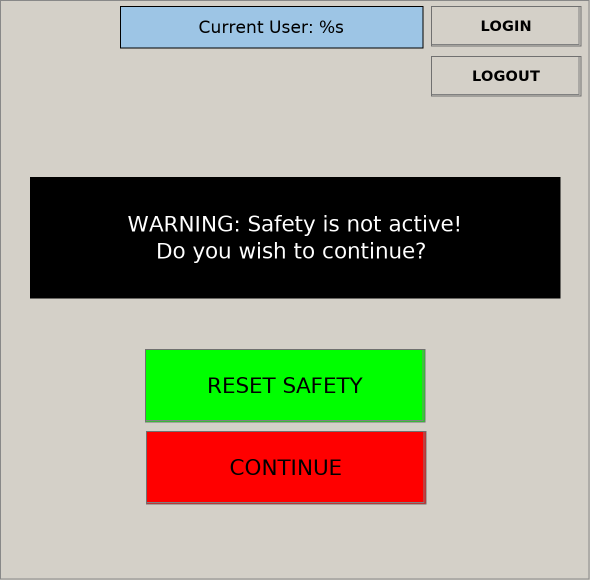
VISUALIZATION safetyDisableWarning  // 590x580
    Rectangle (30,177 530x121), "WARNING: Safety is not active! Do you wish to continue?", text variable: MAIN.sSafetyResetMsg
    Button (145,349 280x73), "RESET SAFETY"
        toggle GVL_machine.bSafetyBypass
    Button (146,431 280x73), "CONTINUE"
        OnMouseDown: change screen: Previous 
        OnMouseDown: execute { main.fbSafetyBypassTim(IN := FALSE); }
    Button (431,6 150x40), "LOGIN"
        OnMouseDown: VisuUserMgmt Type=Login
    Button (431,56 150x40), "LOGOUT"
        OnMouseDown: VisuUserMgmt Type=Logout
    Textfield (120,6 303x42), "Current User: %s", text variable: VisuElems.CurrentUserName
END_VISUALIZATION

// ---- VISUs/VISUs/safetyResetScreen.TcVIS
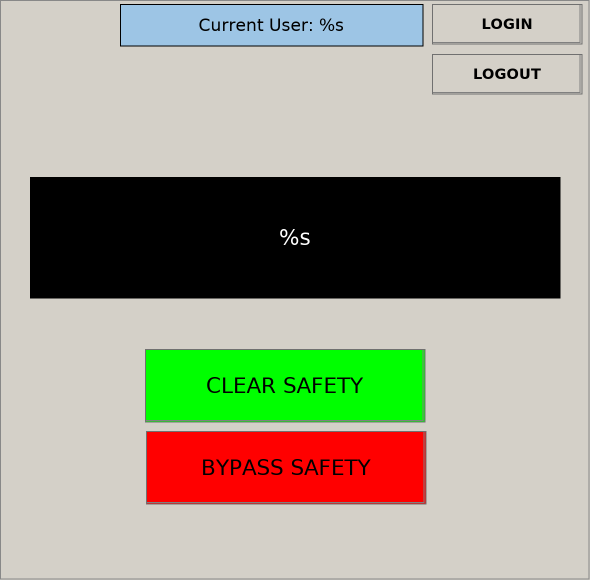
VISUALIZATION safetyResetScreen  // 590x580
    Rectangle (30,177 530x121), "%s", text variable: MAIN.sSafetyResetMsg
    Button (145,349 280x73), "CLEAR SAFETY"
        toggle MAIN.bSafetyResetBtn
    Button (146,431 280x73), "BYPASS SAFETY"
        toggle GVL_machine.bSafetyBypass
        OnMouseDown: execute {
            IF NOT GVL_devices.fbEstop.bEstopSigOk THEN
            	main.bBypassResetEstop := TRUE;
            END_IF
        }
    Button (432,4 150x40), "LOGIN"
        OnMouseDown: VisuUserMgmt Type=Login
    Button (432,54 150x40), "LOGOUT"
        OnMouseDown: VisuUserMgmt Type=Logout
    Textfield (120,4 303x42), "Current User: %s", text variable: VisuElems.CurrentUserName
END_VISUALIZATION

// ---- VISUs/VISUs/settingsScreen.TcVIS
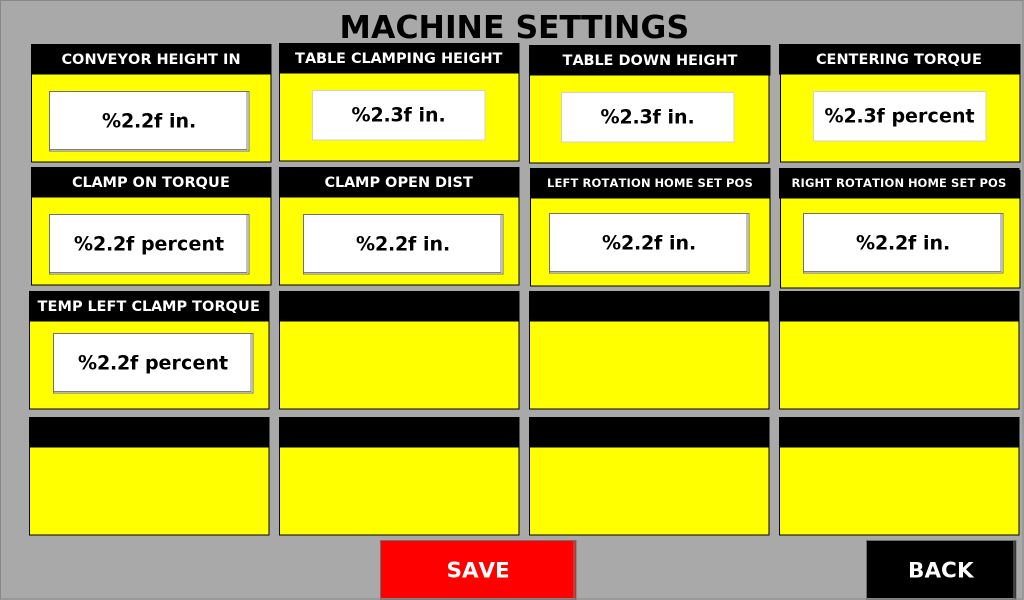
VISUALIZATION settingsScreen  // 1024x600
    RoundedRectangle (29,291 240x118)
    RoundedRectangle (279,43 240x118)
    RoundedRectangle (529,45 240x118)
    RoundedRectangle (29,417 240x118)
    RoundedRectangle (780,44 240x118)
    RoundedRectangle (780,170 240x118)
    RoundedRectangle (530,168 240x118)
    RoundedRectangle (279,291 240x118)
    RoundedRectangle (279,417 240x118)
    Label (183,10 663x34), "MACHINE SETTINGS"
    Textfield (661,76 61x30)
    Textfield (583,76 61x30)
    Textfield (327,202 61x30)
    Textfield (555,75 84x30)
    RoundedRectangle (279,417 240x30)
    RoundedRectangle (279,291 240x30)
    RoundedRectangle (29,291 240x30), "TEMP LEFT CLAMP TORQUE"
    RoundedRectangle (29,417 240x30)
    Textfield (680,76 61x30)
    Textfield (813,91 173x50), "%2.3f percent", text variable: GVL_persistent.fCenteringTorque
        OnMouseClick: write the text variable via VisuDialogs.Numpad
        OnMouseClick: OpenDialog Dialog=VisuDialogs.MessageBox, Parameters={eType: VisuDialogs.MessageBoxDialog_Types.OK, sMessageTxt: GVL_machine.sEditMessage, sTitle: GVL_machine.sEditTitle}, OpenModal=True, OpenCentered=True
        OnMouseClick: execute { GVL_machine.bFlashSaveBtn := TRUE; }
    Textfield (312,90 173x50), "%2.3f in.", text variable: GVL_persistent.fTableClampHeight
        OnMouseClick: write the text variable via VisuDialogs.Numpad
        OnMouseClick: OpenDialog Dialog=VisuDialogs.MessageBox, Parameters={eType: VisuDialogs.MessageBoxDialog_Types.OK, sMessageTxt: GVL_machine.sEditMessage, sTitle: GVL_machine.sEditTitle}, OpenModal=True, OpenCentered=True
        OnMouseClick: execute { GVL_machine.bFlashSaveBtn := TRUE; }
    Textfield (561,92 173x50), "%2.3f in.", text variable: GVL_persistent.fTableDownHeight
        OnMouseClick: write the text variable via VisuDialogs.Numpad
        OnMouseClick: OpenDialog Dialog=VisuDialogs.MessageBox, Parameters={eType: VisuDialogs.MessageBoxDialog_Types.OK, sMessageTxt: GVL_machine.sEditMessage, sTitle: GVL_machine.sEditTitle}, OpenModal=True, OpenCentered=True
        OnMouseClick: execute { GVL_machine.bFlashSaveBtn := TRUE; }
        OnMouseDown: write the text variable via Default
        OnMouseDown: OpenDialog Dialog=VisuDialogs.MessageBox, Parameters={eType: VisuDialogs.MessageBoxDialog_Types.OK, sMessageTxt: GVL_machine.sEditMessage, sTitle: GVL_machine.sEditTitle}, OpenModal=True, OpenCentered=True
    RoundedRectangle (779,291 240x118)
    RoundedRectangle (779,417 240x118)
    Textfield (77,201 61x30)
    RoundedRectangle (779,291 240x30)
    RoundedRectangle (779,417 240x30)
    RoundedRectangle (31,44 240x118)
    RoundedRectangle (31,167 240x118)
    Textfield (78,200 61x30)
    Button (49,91 200x60), "%2.2f in.", text variable: GVL_persistent.fTableConveyorHeight
        OnMouseClick: write the text variable via VisuDialogs.Numpad
        OnMouseClick: OpenDialog Dialog=VisuDialogs.MessageBox, Parameters={eType: VisuDialogs.MessageBoxDialog_Types.OK, sMessageTxt: GVL_machine.sEditMessage, sTitle: GVL_machine.sEditTitle}, OpenModal=True, OpenCentered=True
        OnMouseClick: execute { GVL_machine.bFlashSaveBtn := TRUE; }
    Button (49,214 200x60), "%2.2f percent", text variable: GVL_persistent.fClampOnTorque
        OnMouseClick: write the text variable via VisuDialogs.Numpad
        OnMouseClick: OpenDialog Dialog=VisuDialogs.MessageBox, Parameters={eType: VisuDialogs.MessageBoxDialog_Types.OK, sMessageTxt: GVL_machine.sEditMessage, sTitle: GVL_machine.sEditTitle}, OpenModal=True, OpenCentered=True
        OnMouseClick: execute { GVL_machine.bFlashSaveBtn := TRUE; }
    RoundedRectangle (279,167 240x118)
    Button (303,214 200x60), "%2.2f in.", text variable: GVL_persistent.fClampOpenDist
        OnMouseClick: write the text variable via VisuDialogs.Numpad
        OnMouseClick: OpenDialog Dialog=VisuDialogs.MessageBox, Parameters={eType: VisuDialogs.MessageBoxDialog_Types.OK, sMessageTxt: GVL_machine.sEditMessage, sTitle: GVL_machine.sEditTitle}, OpenModal=True, OpenCentered=True
        OnMouseClick: execute { GVL_machine.bFlashSaveBtn := TRUE; }
    RoundedRectangle (529,291 240x118)
    RoundedRectangle (529,417 240x118)
    RoundedRectangle (529,291 240x30)
    RoundedRectangle (529,417 240x30)
    Button (866,540 150x60), "BACK"
        OnMouseDown: change screen: Previous maintenanceScreen3
    Button (380,540 196x60), "SAVE", colour toggle: GVL_machine.bSaveBtnFlashOn
        OnMouseDown: execute { GVL_machine.bSaveBtn := TRUE; }
    Button (803,213 200x60), "%2.2f in.", text variable: GVL_persistent.fRhtRotationHomePos
        OnMouseClick: write the text variable via VisuDialogs.Numpad
        OnMouseClick: OpenDialog Dialog=VisuDialogs.MessageBox, Parameters={eType: VisuDialogs.MessageBoxDialog_Types.OK, sMessageTxt: GVL_machine.sEditMessage, sTitle: GVL_machine.sEditTitle}, OpenModal=True, OpenCentered=True
        OnMouseClick: execute { GVL_machine.bFlashSaveBtn := TRUE; }
    Button (549,213 200x60), "%2.2f in.", text variable: GVL_persistent.fLftRotationHomePos
        OnMouseClick: write the text variable via VisuDialogs.Numpad
        OnMouseClick: OpenDialog Dialog=VisuDialogs.MessageBox, Parameters={eType: VisuDialogs.MessageBoxDialog_Types.OK, sMessageTxt: GVL_machine.sEditMessage, sTitle: GVL_machine.sEditTitle}, OpenModal=True, OpenCentered=True
        OnMouseClick: execute { GVL_machine.bFlashSaveBtn := TRUE; }
    RoundedRectangle (31,44 240x30), "CONVEYOR HEIGHT IN"
        OnMouseClick: OpenDialog Dialog=VisuDialogs.MessageBox, Parameters={eType: VisuDialogs.MessageBoxDialog_Types.OK, sMessageTxt: GVL_machine.sConvHeightMsg, sTitle: GVL_machine.sDescTitle}, OpenModal=True, OpenCentered=True
    RoundedRectangle (530,168 240x30), "LEFT ROTATION HOME SET POS"
        OnMouseClick: OpenDialog Dialog=VisuDialogs.MessageBox, Parameters={eType: VisuDialogs.MessageBoxDialog_Types.OK, sMessageTxt: GVL_machine.sLftRotHomeSetMsg, sTitle: GVL_machine.sDescTitle}, OpenModal=True, OpenCentered=True
    RoundedRectangle (279,43 240x30), "TABLE CLAMPING HEIGHT"
        OnMouseClick: OpenDialog Dialog=VisuDialogs.MessageBox, Parameters={eType: VisuDialogs.MessageBoxDialog_Types.OK, sMessageTxt: GVL_machine.sClampHeightMsg, sTitle: GVL_machine.sDescTitle}, OpenModal=True, OpenCentered=True
    RoundedRectangle (779,168 240x30), "RIGHT ROTATION HOME SET POS"
        OnMouseClick: OpenDialog Dialog=VisuDialogs.MessageBox, Parameters={eType: VisuDialogs.MessageBoxDialog_Types.OK, sMessageTxt: GVL_machine.sRhtRotHomeSetMsg, sTitle: GVL_machine.sDescTitle}, OpenModal=True, OpenCentered=True
    RoundedRectangle (779,44 240x30), "CENTERING TORQUE"
        OnMouseClick: OpenDialog Dialog=VisuDialogs.MessageBox, Parameters={eType: VisuDialogs.MessageBoxDialog_Types.OK, sMessageTxt: GVL_machine.sCenterTorqueMsg, sTitle: GVL_machine.sDescTitle}, OpenModal=True, OpenCentered=True
    RoundedRectangle (530,45 240x30), "TABLE DOWN HEIGHT"
        OnMouseClick: OpenDialog Dialog=VisuDialogs.MessageBox, Parameters={eType: VisuDialogs.MessageBoxDialog_Types.OK, sMessageTxt: GVL_machine.sDownHeightMsg, sTitle: GVL_machine.sDescTitle}, OpenModal=True, OpenCentered=True
    RoundedRectangle (31,167 240x30), "CLAMP ON TORQUE"
        OnMouseClick: OpenDialog Dialog=VisuDialogs.MessageBox, Parameters={eType: VisuDialogs.MessageBoxDialog_Types.OK, sMessageTxt: GVL_machine.sClampOnTorqueMsg, sTitle: GVL_machine.sDescTitle}, OpenModal=True, OpenCentered=True
    RoundedRectangle (279,167 240x30), "CLAMP OPEN DIST"
        OnMouseClick: OpenDialog Dialog=VisuDialogs.MessageBox, Parameters={eType: VisuDialogs.MessageBoxDialog_Types.OK, sMessageTxt: GVL_machine.sClampOpenDistMsg, sTitle: GVL_machine.sDescTitle}, OpenModal=True, OpenCentered=True
    Button (53,333 200x60), "%2.2f percent", text variable: GVL_persistent.fTempLftClampTorque
        OnMouseClick: write the text variable via VisuDialogs.Numpad
        OnMouseClick: OpenDialog Dialog=VisuDialogs.MessageBox, Parameters={eType: VisuDialogs.MessageBoxDialog_Types.OK, sMessageTxt: GVL_machine.sEditMessage, sTitle: GVL_machine.sEditTitle}, OpenModal=True, OpenCentered=True
        OnMouseClick: execute { GVL_machine.bFlashSaveBtn := TRUE; }
END_VISUALIZATION
